Staubli VAL3: iTool.pgx

public program iTool(num& nNum[] (dimensions=1))
begin
  nNum=dioGet(iIdent1)+(2*dioGet(iIdent2))+(4*dioGet(iIdent3))
end
